TYPE SystemControl :
STRUCT
	StartUpRequest : BOOL;
	ShutdownRequest : BOOL;
	Reset : BOOL;
END_STRUCT
END_TYPE

(* stored: Version 1.1.0.1
   DUT SystemControl: Id {0f073b3a-007f-4a3f-97c8-6376fc135e34} *)
